INTERFACE IACComponent EXTENDS IACObject

PROPERTY ACIdentifier : STRING
GET
END_GET
END_PROPERTY

PROPERTY Childs : ARRAY [1..GCL.cChildsMAX] OF IACComponent
GET
END_GET
END_PROPERTY

METHOD FB_childinit
VAR_INPUT
END_VAR
END_METHOD

METHOD FindChildOfTypeAt : IACComponent
VAR_INPUT
	atIndex : INT;
	objectType : TypeOfACObjectEnum;
	maxChildDepth : INT;
END_VAR
END_METHOD

METHOD FindChildsOfType
VAR_INPUT
	objectType : TypeOfACObjectEnum;
	maxChildDepth : INT;
END_VAR
VAR_IN_OUT
	result : ARRAY [0..GCL.cChildsMAX] OF IACComponent;
END_VAR
END_METHOD

METHOD FindObjectByID : IACObject
VAR_INPUT
	instanceID : UDINT;
END_VAR
END_METHOD

METHOD FindParentOfType : IACComponent
VAR_INPUT
	objectType : TypeOfACObjectEnum;
END_VAR
END_METHOD

PROPERTY Parent : IACComponent
GET
END_GET
END_PROPERTY

PROPERTY Root : IACVariobatch
GET
END_GET
END_PROPERTY

METHOD RunMain : BOOL
VAR_INPUT
END_VAR
END_METHOD

END_INTERFACE

(* stored: Version 1.1.0.1, ProductVersion 3.1.4024.6
   Itf IACComponent: Id {aa5db2de-8e30-44bc-a2ed-e07801df9b40}
   Property ACIdentifier: Id {4a6a2e30-067c-412e-a072-129bdd94b48c}
   Get Get: Id {8169ae38-840f-42fb-ba55-225e10fd2986}
   Property Childs: Id {5e0de931-5dcf-4a48-b8de-988e6265bfad}
   Get Get: Id {0067385c-aec5-46e0-9861-5598154b513b}
   Method FB_childinit: Id {943c996b-1b40-428b-9a8a-7fed8d62eefc}
   Method FindChildOfTypeAt: Id {3bc8339f-b19a-41c0-8a8b-12a6e18a9419}
   Method FindChildsOfType: Id {acc1bbbd-abbe-4339-b638-c2c7ccab0c75}
   Method FindObjectByID: Id {4b83826e-e613-4eb2-9e79-b63bf8b8b54f}
   Method FindParentOfType: Id {e0c02f3b-7a29-4316-8910-aadd9b0e7843}
   Property Parent: Id {64ce908b-a3ca-418e-9949-0ba5b598ca74}
   Get Get: Id {8f59059a-e136-49d9-9df1-b677a13e4981}
   Property Root: Id {4192da07-8975-42a9-b8cd-9be60369dea6}
   Get Get: Id {848ed9f2-bd8a-400d-9393-11c92b3a092d}
   Method RunMain: Id {c7be0c22-6c28-4b26-8ac8-b59603486301} *)
